// Reads a length for length-delimited data.
FUNCTION F_ParseLength : HRESULT
VAR_IN_OUT      
    stCtx : ST_ParseContext;
END_VAR
VAR_OUTPUT
    nLength : UDINT;
END_VAR


F_ParseLength := F_ParseRawVarint32(stCtx, nLength);

END_FUNCTION

(* stored: Version 1.1.0.1
   POU F_ParseLength: Id {93c884db-4f4d-492d-b48f-8e5fbd80cd44}, SpecialFunc None *)
